FUNCTION_BLOCK TcMessage_Ext IMPLEMENTS ITcMessage_Ext
VAR_INPUT
END_VAR
VAR_OUTPUT
END_VAR
VAR
    fbMsg : FB_TcMessage; 
	_loggerLevel : TcEventSeverity := TcEventSeverity.Info;
END_VAR

PROPERTY PUBLIC LoggerLevel : TcEventSeverity
GET
LoggerLevel := _loggerLevel;
END_GET
SET
_loggerLevel := LoggerLevel;
END_SET
END_PROPERTY

METHOD PUBLIC Send : BOOL
VAR_INPUT
	eventType : Tc3_EventLogger.TcEventEntry;
	args : STRING(255);
END_VAR
IF eventType.eSeverity >= LoggerLevel THEN
	THIS^.fbMsg.CreateEx(eventType, 0);
	THIS^.fbMsg.ipArguments.AddString(args);
	THIS^.fbMsg.Send(0);
	THIS^.fbMsg.Release();
END_IF
END_METHOD

END_FUNCTION_BLOCK

(* stored: Version 1.1.0.1, ProductVersion 3.1.4024.12
   POU TcMessage_Ext: Id {3f852920-143f-462f-9e3f-f9ba6d6e0946}, SpecialFunc None
   Property LoggerLevel: Id {d56fe456-719d-4a96-8c1d-a040859bbf48}
   Get Get: Id {3fda9917-8d32-4dd1-862a-7a10160231fe}
   Set Set: Id {73004715-4d1a-4abc-9f0d-67258850f9eb}
   Method Send: Id {695ccdb3-d080-4ce2-9eb6-6d31e250fe47} *)
